FUNCTION_BLOCK FB_SerialCom
VAR_IN_OUT
	TxBuffer	: ComBuffer;
	RxBuffer	: ComBuffer;
	eReceiveErrorID	: ComError_t;
END_VAR
VAR
	fbReceive		: ReceiveData;
	nReceiveCounter	: UDINT;
	prefix : ARRAY[0..1] OF BYTE;
	receivedata : ARRAY [0..15] OF BYTE;
	packet_ID : BYTE := 37;
	packet_length : BYTE := 12;	
	
	crc : WORD;
	crc_check : WORD;
	pt_crc : POINTER TO WORD;
	crc12 : ARRAY [0..1] OF BYTE;	
	dataArray : ARRAY[0..11] OF BYTE;
	i : USINT;
	acc_x : ARRAY [0..3] OF BYTE;
	acc_y : ARRAY [0..3] OF BYTE;
	acc_z : ARRAY [0..3] OF BYTE;
	pt_x : POINTER TO REAL;
    x_acc : REAL;
	pt_y : POINTER TO REAL;
    y_acc : REAL;
	pt_z : POINTER TO REAL;
    z_acc : REAL;
END_VAR

prefix[0] := packet_ID;
prefix[1] := packet_length;

fbReceive(
	RXbuffer:= RxBuffer,
	pPrefix := ADR(prefix),
	LenPrefix := 2,
	pReceiveData := ADR(receivedata),
	SizeReceiveData  := 16,								
	Error=> ,
	DataReceived=>,
		);
IF fbReceive.Error <> COMERROR_NOERROR THEN
	eReceiveErrorID := fbReceive.Error;
END_IF
IF fbReceive.DataReceived THEN							
	nReceiveCounter := nReceiveCounter + 1;
END_IF

doCRC16Check1();

METHOD doCRC16Check1 : BOOL
VAR_INPUT
END_VAR
FOR i:=0 TO 11 DO
	dataArray[i] := receivedata[i+4];
END_FOR


crc := F_DATA_TO_CRC16_CCITT(
	pData := ADR(dataArray),
	cbData := BYTE_TO_UDINT(packet_length),
	crc := 16#FFFF);

crc12[0] := receivedata[2];
crc12[1] := receivedata[3];
pt_crc := ADR(crc12);
crc_check := pt_crc^;
END_METHOD

PROPERTY getAccelerationValueX : REAL
GET
IF crc_check = crc THEN

	acc_x[0] := receivedata[4];
	acc_x[1] := receivedata[5];
	acc_x[2] := receivedata[6];
	acc_x[3] := receivedata[7];
	pt_x := ADR(acc_x);
	x_acc := pt_x^;
END_IF

getAccelerationValueX := x_acc;
END_GET
END_PROPERTY

PROPERTY getAccelerationValueY : REAL
GET
IF crc_check = crc THEN
	
	acc_y[0] := receivedata[8];
	acc_y[1] := receivedata[9];
	acc_y[2] := receivedata[10];
	acc_y[3] := receivedata[11];
	pt_y := ADR(acc_y);
	y_acc := pt_y^;

END_IF
getAccelerationValueY := y_acc;
END_GET
END_PROPERTY

PROPERTY getAccelerationValueZ : REAL
GET
IF crc_check = crc THEN
	
	acc_z[0] := receivedata[12];
	acc_z[1] := receivedata[13];
	acc_z[2] := receivedata[14];
	acc_z[3] := receivedata[15];
	pt_z := ADR(acc_z);
	z_acc := pt_z^;
END_IF

getAccelerationValueZ := z_acc;
END_GET
END_PROPERTY

END_FUNCTION_BLOCK

(* stored: Version 1.1.0.1, ProductVersion 3.1.4024.12
   POU FB_SerialCom: Id {181e7c70-138b-446a-a6f5-34e588388885}, SpecialFunc None
   Method doCRC16Check1: Id {402d79e6-a8fb-4a7c-8d55-db08bc01f1c2}
   Property getAccelerationValueX: Id {bc94098a-9a77-45c6-908e-086ed4a9c91b}
   Get Get: Id {ba6ddbbc-cc5d-417a-8cf7-c48fe0e1a0b2}
   Property getAccelerationValueY: Id {bf4e2282-4810-4b14-b6bd-6cc9d8487ce8}
   Get Get: Id {5a78a6f3-4b22-4600-9d01-dc7af91cccc7}
   Property getAccelerationValueZ: Id {7c40e5c6-9f5b-49d3-8d6e-7d9c99c30b17}
   Get Get: Id {82b17f14-e3c3-4811-8412-1ca005785c16} *)
